Staubli VAL3: takestop.pgx

program takestop()
begin
  //信号
  b2=true
  while true
    if distop==true
      call stop()
      b2=true
    endIf
    if distart==true
      if b2
        call Message("启动...",true)
      endIf
      b2=false
    endIf

    //    wait(distop==true)
    //    b2=true

    //    wait(distart==true)
    //    b2=false

    delay(0)
  endWhile
end
